ABB RobotStudio station: plantilla - pruebas_20220202-080609.rsstn

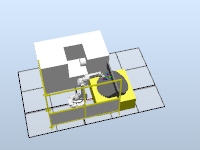
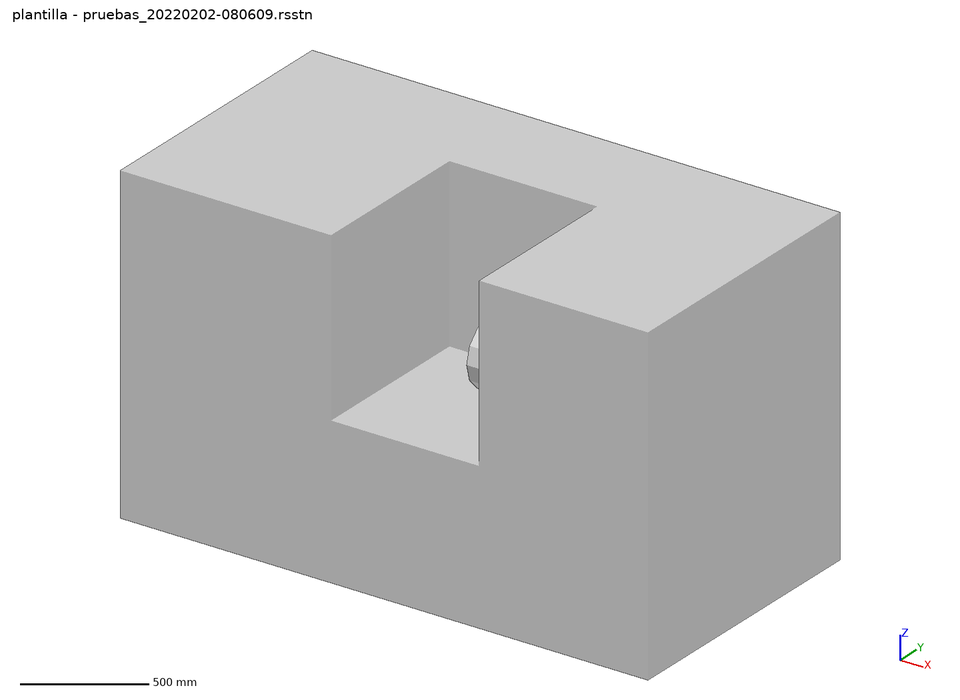
[picture v1: parts stored in the station drawn from their meshes, with robot base, taught points and paths (robot models come from the ABB library and are not in the file)]
Station Station (saved by RobotStudio 21.2.9526.0)
Layout (positions relative to the parent item):
  - IRB1660ID_4_155__03 [mechanism, from Robots\IRB1660ID_4_155__03.rslib] at (0, 0, 0) mm; joint values [0, 0, 0, 0, 0.5236, 0] (rad or m)
  - Pinza_1 [mechanism, from Efectores_finales - Copy\PinzaF_1.rslib] at (944.87, 0, 1229) mm, rotated rx 180 ry 60 rz 180 deg; joint values [0, 0] (rad or m)
  - Pinza_2 [mechanism, from Efectores_finales - Copy\PinzaF_2.rslib] at (944.87, 0, 1229) mm, rotated rx 180 ry 60 rz 180 deg; joint values [0, 0] (rad or m)
  - Torno [part] at (-1172.42, 1966.27, 0) mm, rotated rx 0 ry 0 rz 180 deg, size 2500 x 1300 x 1500 mm
  - Fence_740 [graphiccomponentgroup, from Equipment\Fence_740.rslib] at (-1160.76, -802.49, 0) mm
    - Body 1 [part, from Equipment\Fence_740.rslib]
    - Body 2 [part, from Equipment\Fence_740.rslib]
  - Fence_2500 [graphiccomponentgroup, from Equipment\Fence_2500.rslib] at (1297.15, -826.85, 0) mm, rotated rx 0 ry 0 rz 90 deg
    - Body 1 [part, from Equipment\Fence_2500.rslib]
    - Body 2 [part, from Equipment\Fence_2500.rslib]
  - Fence_740_2 [graphiccomponentgroup, from Equipment\Fence_740.rslib] at (-1148.66, -57.63, 0) mm
    - Body 1 [part, from Equipment\Fence_740.rslib]
    - Body 2 [part, from Equipment\Fence_740.rslib]
  - Portapiezas [mechanism] at (0, 0, 0) mm; joint values [0] (rad or m)
      links: L1, L2
Attachment: Pinza_1 is attached to IRB1660ID_4_155__03 / Link6
Attachment: Pinza_2 is attached to IRB1660ID_4_155__03 / Link6
Targets, tools, work objects and paths stored in the station, written as RAPID:
! task (no controller)
MODULE CalibData
  PERS tooldata Pinza_1:=[TRUE,[[-100,0,70],[0.707106781,0,-0.707106781,0]],[1,[0,0,1],[1,0,0,0],0,0,0]];
  PERS tooldata Vara:=[TRUE,[[0,0,250],[0.707106781,0,0,0.707106781]],[1,[0,0,1],[1,0,0,0],0,0,0]];
  PERS tooldata Soplador:=[TRUE,[[0,-70,70],[0.5,0.5,-0.5,0.5]],[1,[0,0,1],[1,0,0,0],0,0,0]];
  PERS tooldata Pinza_2_1:=[TRUE,[[100,0,70],[0.707106781,0,0.707106781,0]],[1,[0,0,2],[1,0,0,0],0,0,0]];
ENDMODULE

